PROGRAM DLOG_FILE_CSV_DEMO
VAR
	RTC_2: RTC_2;
	x : DLOG_DATA;
	DLOG_STORE_FILE_CSV : DLOG_STORE_FILE_CSV;
	CLK_PRG: CLK_PRG;
	cur_dt: DT;
	enable: BOOL;
	rtc_set : BOOL := TRUE;

	trig_t : UDINT := 0;
	trig_m : BOOL;

	x1: DLOG_DT;
	x2 : DLOG_REAL;
	x3 : DLOG_DINT;
	x4 : DLOG_BOOL;
	x5: DLOG_STRING;
	GEN_SIN_1: GEN_SIN;
	COUNT_DR: COUNT_DR;
	error_c: DWORD;
	error_t: BYTE;
END_VAR

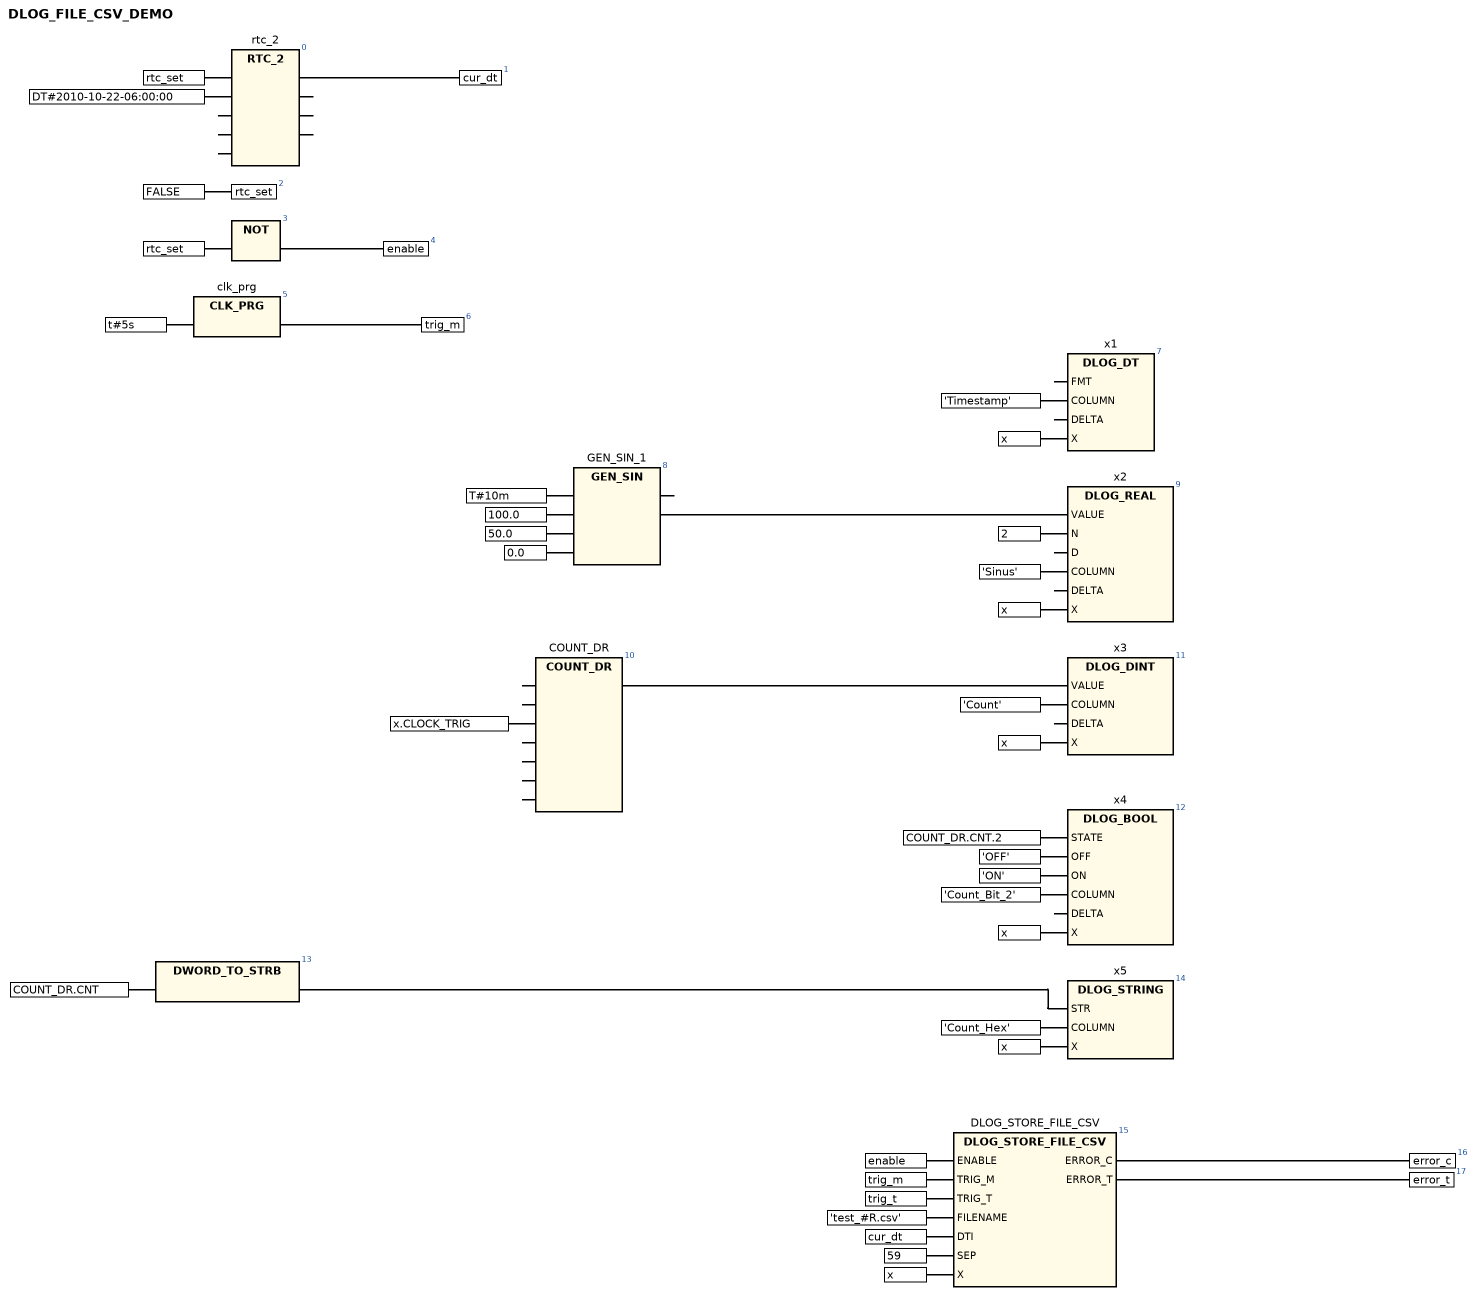
rtc_2(_in1 := rtc_set, _in2 := DT#2010-10-22-06:00:00);
cur_dt := rtc_2._out1;
rtc_set := FALSE;
enable := NOT rtc_set;
clk_prg(_in1 := t#5s);
trig_m := clk_prg._out1;
x1(COLUMN := 'Timestamp', X := x); // DLOG_DT
GEN_SIN_1(_in1 := T#10m, _in2 := 100.0, _in3 := 50.0, _in4 := 0.0); // GEN_SIN
x2(VALUE := GEN_SIN_1._out2, N := 2, COLUMN := 'Sinus', X := x); // DLOG_REAL
COUNT_DR(_in3 := x.CLOCK_TRIG);
x3(VALUE := COUNT_DR._out1, COLUMN := 'Count', X := x); // DLOG_DINT
x4(STATE := COUNT_DR.CNT.2, OFF := 'OFF', ON := 'ON', COLUMN := 'Count_Bit_2', X := x); // DLOG_BOOL
x5(STR := DWORD_TO_STRB(COUNT_DR.CNT), COLUMN := 'Count_Hex', X := x); // DLOG_STRING
DLOG_STORE_FILE_CSV(
    ENABLE := enable,
    TRIG_M := trig_m,
    TRIG_T := trig_t,
    FILENAME := 'test_#R.csv',
    DTI := cur_dt,
    SEP := 59,
    X := x);
error_c := DLOG_STORE_FILE_CSV.ERROR_C;
error_t := DLOG_STORE_FILE_CSV.ERROR_T;

END_PROGRAM

(* stored: Version 1.1.0.1, ProductVersion 3.1.4022.7
   POU DLOG_FILE_CSV_DEMO: Id {a630463b-80f9-4151-9f72-4e244b2512ec}, SpecialFunc None *)
